SUBAPPLICATION Uebung_039_sub_Outputs_AX (* Spiegelabfolge V2 mit Schrittkette SUB Out *)
  (* Standard: 61499-2; Description: Copyright (c) 2023 Meisterschulen am Ostbahnhof This program and the accompanying materials are made available under the terms of the Eclipse Public License 2.0 which is available at https://www.eclipse.org/legal/epl-2.0/ SPDX-License-Identifier: EPL-2.0 *)
  (* Version 1.0, 2024-03-03, Franz Höpfinger, Meisterschulen am Ostbahnhof, initial API and implementation and/or initial documentation *)
  PACKAGE Uebungen;
  IMPORT isobus::UT::Q::const::IDs::ID_NULL;
  IMPORT logiBUS::io::DQ::logiBUS_DO;
  IMPORT logiBUS::io::DQ::logiBUS_DO_S;
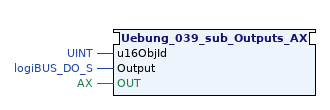
  VAR_INPUT
    u16ObjId : UINT := ID_NULL; (* Object ID Softkey/Button *)
    Output : logiBUS::io::DQ::logiBUS_DO_S := logiBUS_DO::Invalid;
  END_VAR
  SOCKETS
    OUT : adapter::types::unidirectional::AX;
  END_SOCKETS
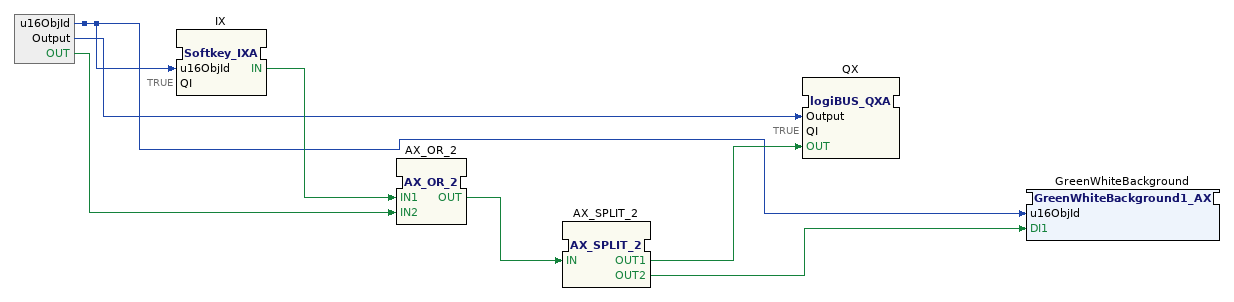
  FBS
    QX : logiBUS::io::DQ::logiBUS_QXA(QI := TRUE);
    IX : isobus::UT::io::Softkey::Softkey_IXA(QI := TRUE);
    AX_OR_2 : adapter::booleanOperators::AX_OR_2;
    AX_SPLIT_2 : adapter::events::unidirectional::AX_SPLIT_2;
  END_FBS
  SUBAPPS
    GreenWhiteBackground : MyLib::sys::GreenWhiteBackground1_AX;
  END_SUBAPPS
  DATA_CONNECTIONS
    u16ObjId TO GreenWhiteBackground.u16ObjId;
    u16ObjId TO IX.u16ObjId;
    Output TO QX.Output;
  END_CONNECTIONS
  ADAPTER_CONNECTIONS
    AX_SPLIT_2.OUT1 TO QX.OUT;
    IX.IN TO AX_OR_2.IN1;
    AX_SPLIT_2.OUT2 TO GreenWhiteBackground.DI1;
    AX_OR_2.OUT TO AX_SPLIT_2.IN;
    OUT TO AX_OR_2.IN2;
  END_CONNECTIONS
END_SUBAPPLICATION
